(* Schneider Machine Expert - Basic project IC Flashing TM221CE40T, file version 2.7.0.0 *)
(* ProjectInformations: Name=New project *)

HARDWARE
  Cpu 0: TM221CE40T
  ModuleExtensionObject 0: TM3DI32K
  ModuleExtensionObject 1: TM3DQ32TK
  EthernetConfiguration: NetworkName=M221, IpAllocationMode=FixedAddress, IpAddress=192.168.0.2, SubnetMask=255.255.255.0
  SerialLineConfiguration: Baud=Baud19200, Parity=ParityEven, DataBits=DataBits8, StopBits=StopBits1, PhysicalMedium=PhysicalMediumRs485, TransmissionMode=TransmissionModeModbusRtu, SlaveId=1, Addressing=SlaveAddressing
  MastTask: UsePeriodScanMode=false, PeriodScan=100
  FastTask: Period=255
  CpuBehavior: StartingMode=StartAsPreviousState, AutoSaveRamOnEeprom=true, WatchdogPeriod=250

SYMBOLS  (address, symbol, comment, settings)
  %MW100:X14 TL_GREEN  "IO Output"
  %MW100:X15 TL_RED  "IO Output"
  %MW101:X1 BUZZER  "Output"
  %MW0:X4   ROBOT_PAUSE  "Input Robot1"
  %MW1:X6   IVACUM1  "Input Robot2"
  %M0         "M_START"
  %M1         "M_STOP"
  %M2         "M_CONTINUE"
  %M3         "M_PAUSE"
  %M4         "GRIPPER_ROTATE_CLOSE"
  %M5         "STATUS CB ON"
  %M6         "RELEASE_C_GRIPPER"
  %M7         "Reset"
  %M8         "Done"
  %M9         "Trig"
  %M10        "Start Read"
  %M11        "Start"
  %M12        "MANUAL"
  %M13        "Busy"
  %M14        "CB_RT"
  %M15        "DELAY_CUT_LEFT"
  %M16        "Cut Left"
  %M17        "Cut Right"
  %M19        "AUX_Seq_INIT"
  %M20        "Start_Write"
  %M21        "Abort"
  %M22        "Done_Write"
  %M23        "Busy_Write"
  %M24        "Aborted"
  %M25        "Error"
  %M26      MANUAL_GRIP_CLOSE  "M_Q4"
  %M27      SLIDER  "M_Q5"
  %M28        "M_Q6"
  %M29        "Manual Bowl"
  %M30        "EMG_Memory"
  %M31        "Start_Memory"
  %M47        "M_EMG"
  %M49        "POLARITY CHECKED"
  %M50        "NEGATIVE"
  %M51        "POSITIVE"
  %M52        "FIRST RUN"
  %M53        "DONE CUTTING"
  %M54        "NEGATIVE READY"
  %M55        "TRIGGER"
  %M56        "COUNTER OUTPUT"
  %M100       "Abort"
  %M102       "M_START"
  %S4       SB_TB10MS  "Time base of 10 ms generated by an internal clock"
  %S6       SB_TB1S  "Time base of 1 s generated by an internal clock"
  %MW0        "Input Robot1"
  %MW1        "Input Robot2"
  %MW100      "IO Output"
  %MW101      "Output"
  %TM2        "Left Cut"  [Preset=10, Base=TenMilliSeconds]
  %READ_VAR1   "READ OUTPUT ROBOT"  [Link(Value(FBComLinkParameterEnums=EthernetLink)), RemoteDeviceId(Value(int=1)), Timeout(Value(int=100)), ObjType(Value(FBComObjTypeParameterEnums=IW)), FirstObj(Value(int=31)), Quantity(Value(int=2)), IndexData(Value(int=100))]
  %WRITE_VAR0   [Link(Value(FBComLinkParameterEnums=EthernetLink)), RemoteDeviceId(Value(int=1)), Timeout(Value(int=100)), ObjType(Value(FBComObjTypeParameterEnums=MW)), FirstObj(Value(int=31)), Quantity(Value(int=2)), IndexData(Value(int=0))]
  %I0.0       "EMG"
  %I0.1       "PB START"
  %I0.2       "PB STOP"
  %I0.3       "PB Continue"
  %I0.4       "PB Pause"
  %I0.5       "Safety Relay"
  %I0.6       "Homing Sensor 1"
  %I0.7       "Homing Sensor 2"
  %I0.23      "iVacum1"
  %Q0.14      "TL Green"
  %Q0.15      "TL YelloW"
  %Q2.0       "TL Red"
  %Q2.1       "BUZZER"
  %Q2.2       "PB GREEN_LAMP"
  %Q2.3       "PB YELLOW_LAMP"
  %Q2.4       "PB RED_LAMP"

POU New POU
  (* SectionNumber=1 *)

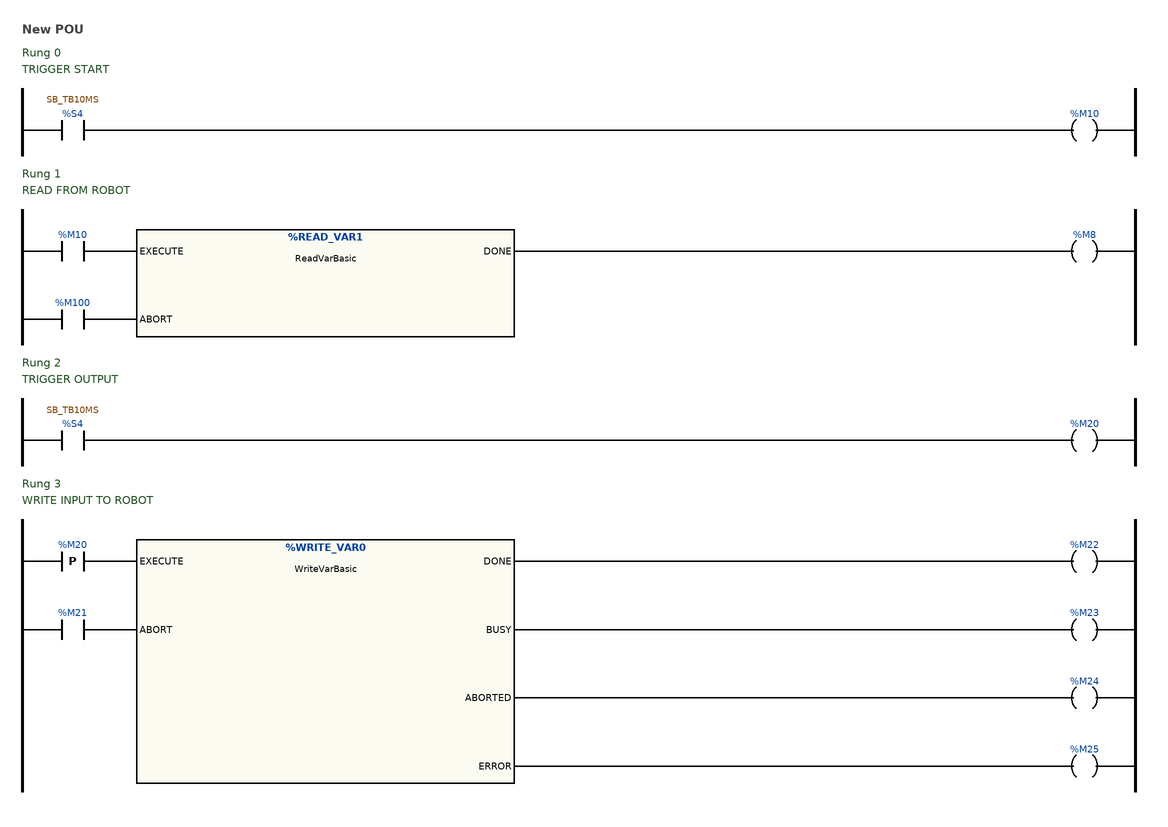

// Rung 0
// TRIGGER START
  LD %S4                  (* SB_TB10MS *)
  ST %M10
  // as ST:
  //   %M10 := SB_TB10MS;

// Rung 1
// READ FROM ROBOT
  BLK %READ_VAR1
  LD %M10
  EXECUTE
  LD %M100
  ABORT
  OUT_BLK
  LD DONE
  ST %M8
  END_BLK
  // as ST:
  //   %READ_VAR1(EXECUTE := %M10, ABORT := %M100);
  //   %M8 := %READ_VAR1.DONE;

// Rung 2
// TRIGGER OUTPUT
  LD %S4                  (* SB_TB10MS *)
  ST %M20
  // as ST:
  //   %M20 := SB_TB10MS;

// Rung 3
// WRITE INPUT TO ROBOT
  BLK %WRITE_VAR0
  LDR %M20
  EXECUTE
  LD %M21
  ABORT
  OUT_BLK
  LD DONE
  ST %M22
  LD BUSY
  ST %M23
  LD ABORTED
  ST %M24
  LD ERROR
  ST %M25
  END_BLK
  // as ST:
  //   %WRITE_VAR0(EXECUTE := RISING(%M20), ABORT := %M21);
  //   %M22 := %WRITE_VAR0.DONE;
  //   %M23 := %WRITE_VAR0.BUSY;
  //   %M24 := %WRITE_VAR0.ABORTED;
  //   %M25 := %WRITE_VAR0.ERROR;

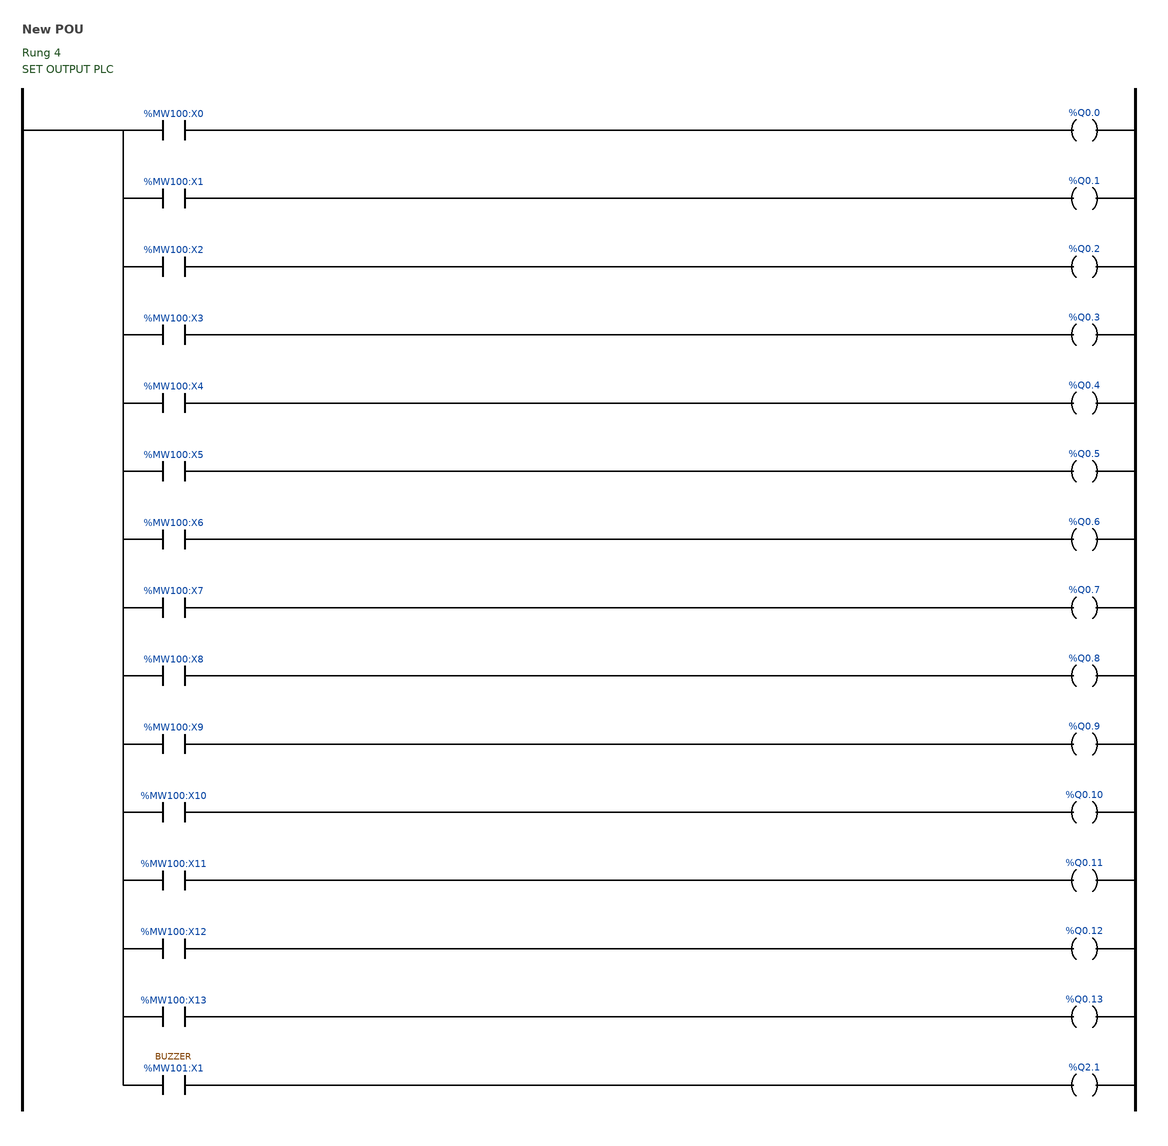

// Rung 4
// SET OUTPUT PLC
  LD 1
  MPS
  AND %MW100:X0
  ST %Q0.0
  MRD
  AND %MW100:X1
  ST %Q0.1
  MRD
  AND %MW100:X2
  ST %Q0.2
  MRD
  AND %MW100:X3
  ST %Q0.3
  MRD
  AND %MW100:X4
  ST %Q0.4
  MRD
  AND %MW100:X5
  ST %Q0.5
  MRD
  AND %MW100:X6
  ST %Q0.6
  MRD
  AND %MW100:X7
  ST %Q0.7
  MRD
  AND %MW100:X8
  ST %Q0.8
  MRD
  AND %MW100:X9
  ST %Q0.9
  MRD
  AND %MW100:X10
  ST %Q0.10
  MRD
  AND %MW100:X11
  ST %Q0.11
  MRD
  AND %MW100:X12
  ST %Q0.12
  MRD
  AND %MW100:X13
  ST %Q0.13
  MPP
  AND %MW101:X1
  ST %Q2.1
  // as ST:
  //   %Q0.0 := %MW100:X0;
  //   %Q0.1 := %MW100:X1;
  //   %Q0.2 := %MW100:X2;
  //   %Q0.3 := %MW100:X3;
  //   %Q0.4 := %MW100:X4;
  //   %Q0.5 := %MW100:X5;
  //   %Q0.6 := %MW100:X6;
  //   %Q0.7 := %MW100:X7;
  //   %Q0.8 := %MW100:X8;
  //   %Q0.9 := %MW100:X9;
  //   %Q0.10 := %MW100:X10;
  //   %Q0.11 := %MW100:X11;
  //   %Q0.12 := %MW100:X12;
  //   %Q0.13 := %MW100:X13;
  //   %Q2.1 := %MW101:X1;

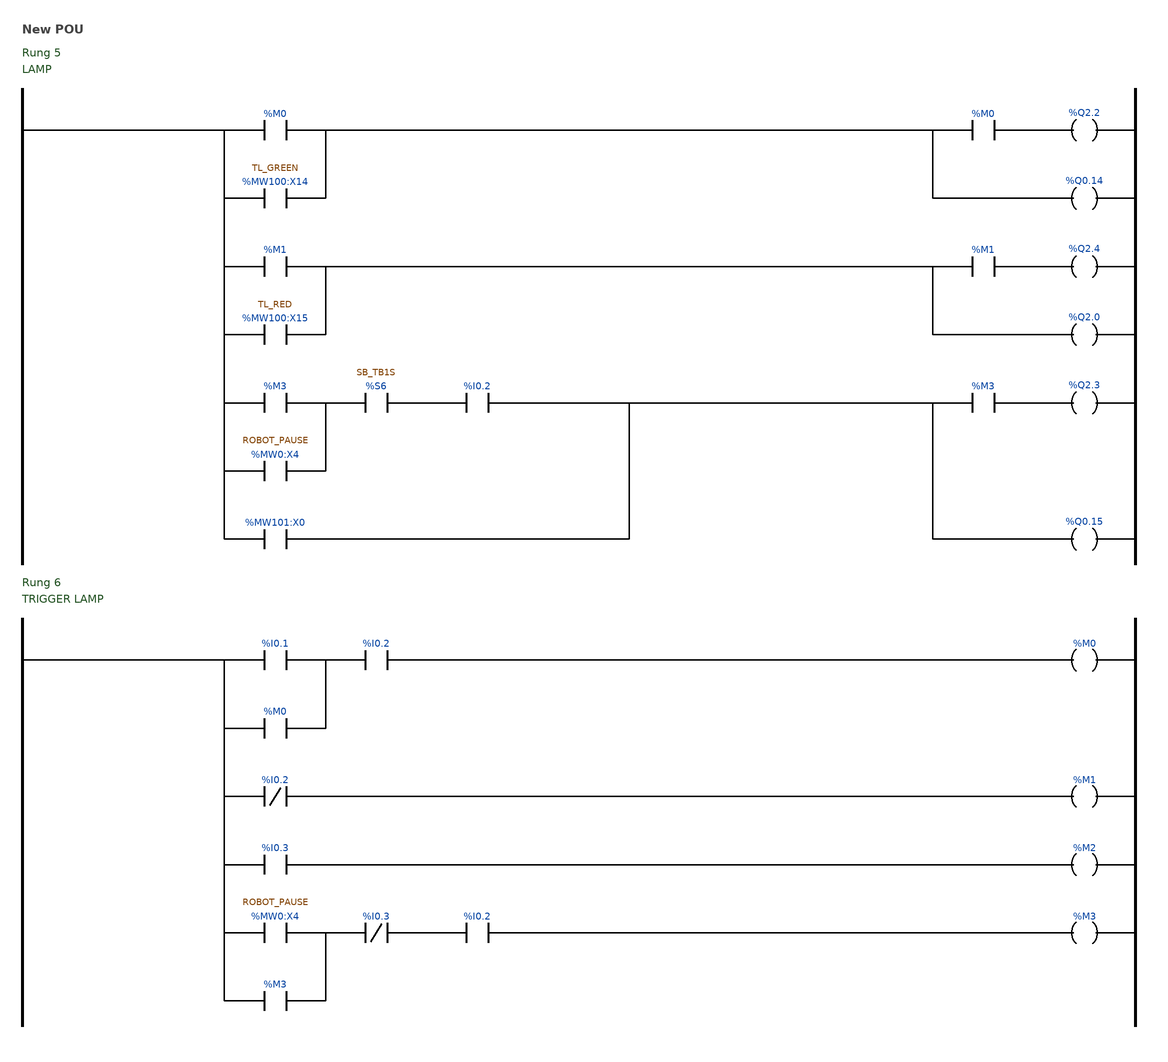

// Rung 5
// LAMP
  LD 1
  MPS
  AND( %M0
  OR %MW100:X14
  )
  MPS
  AND %M0
  ST %Q2.2
  MPP
  ST %Q0.14
  MRD
  AND( %M1
  OR %MW100:X15
  )
  MPS
  AND %M1
  ST %Q2.4
  MPP
  ST %Q2.0
  MPP
  AND( %M3
  OR %MW0:X4
  AND %S6                 (* SB_TB1S *)
  AND %I0.2
  OR %MW101:X0
  )
  MPS
  AND %M3
  ST %Q2.3
  MPP
  ST %Q0.15
  // as ST:
  //   %Q2.2 := (%M0 OR %MW100:X14) AND %M0;
  //   %Q0.14 := %M0 OR %MW100:X14;
  //   %Q2.4 := (%M1 OR %MW100:X15) AND %M1;
  //   %Q2.0 := %M1 OR %MW100:X15;
  //   %Q2.3 := ((%M3 OR %MW0:X4) AND SB_TB1S AND %I0.2 OR %MW101:X0) AND %M3;
  //   %Q0.15 := (%M3 OR %MW0:X4) AND SB_TB1S AND %I0.2 OR %MW101:X0;

// Rung 6
// TRIGGER LAMP
  LD 1
  MPS
  AND( %I0.1
  OR %M0
  )
  AND %I0.2
  ST %M0
  MRD
  ANDN %I0.2
  ST %M1
  MRD
  AND %I0.3
  ST %M2
  MPP
  AND( %MW0:X4
  OR %M3
  )
  ANDN %I0.3
  AND %I0.2
  ST %M3
  // as ST:
  //   %M0 := (%I0.1 OR %M0) AND %I0.2;
  //   %M1 := NOT %I0.2;
  //   %M2 := %I0.3;
  //   %M3 := (%MW0:X4 OR %M3) AND NOT %I0.3 AND %I0.2;

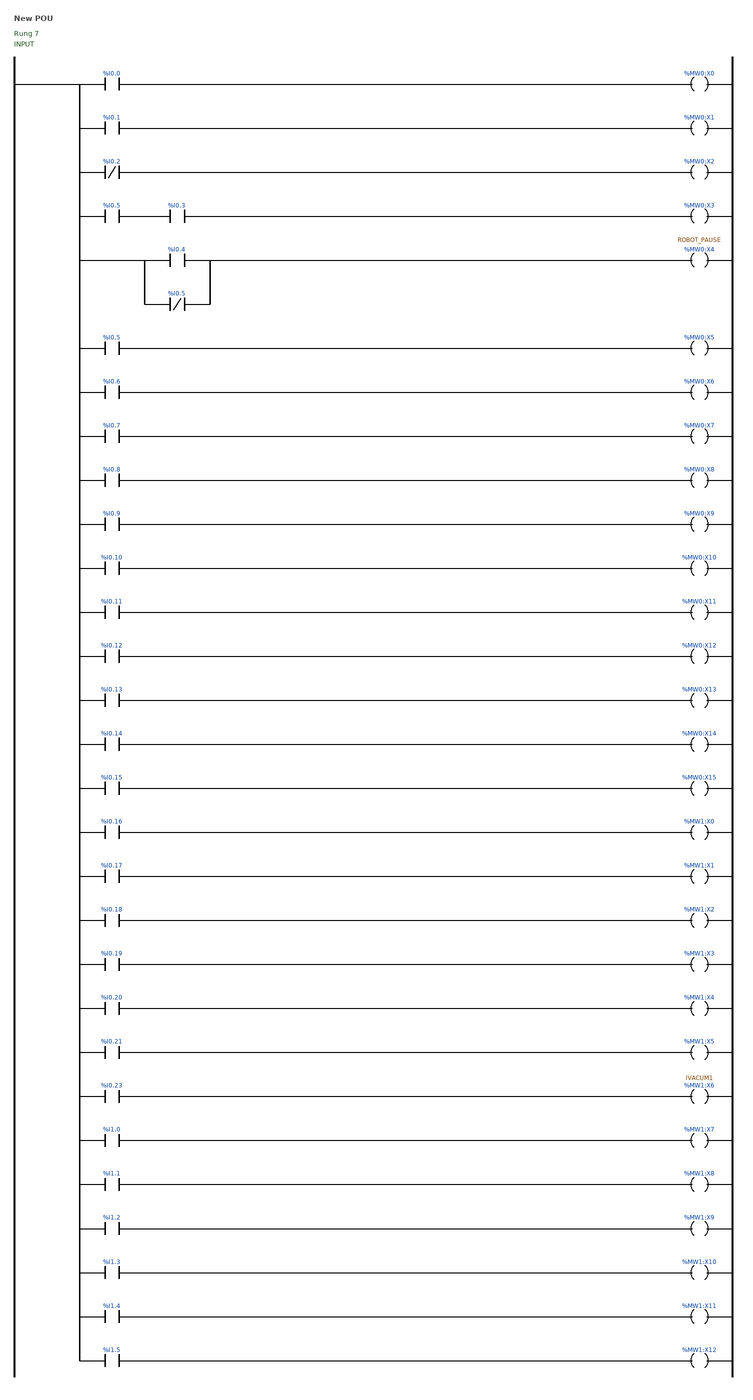

// Rung 7
// INPUT
  LD 1
  MPS
  AND %I0.0
  ST %MW0:X0
  MRD
  AND %I0.1
  ST %MW0:X1
  MRD
  ANDN %I0.2
  ST %MW0:X2
  MRD
  AND %I0.5
  AND %I0.3
  ST %MW0:X3
  MRD
  AND( %I0.4
  ORN %I0.5
  )
  ST %MW0:X4
  MRD
  AND %I0.5
  ST %MW0:X5
  MRD
  AND %I0.6
  ST %MW0:X6
  MRD
  AND %I0.7
  ST %MW0:X7
  MRD
  AND %I0.8
  ST %MW0:X8
  MRD
  AND %I0.9
  ST %MW0:X9
  MRD
  AND %I0.10
  ST %MW0:X10
  MRD
  AND %I0.11
  ST %MW0:X11
  MRD
  AND %I0.12
  ST %MW0:X12
  MRD
  AND %I0.13
  ST %MW0:X13
  MRD
  AND %I0.14
  ST %MW0:X14
  MRD
  AND %I0.15
  ST %MW0:X15
  MRD
  AND %I0.16
  ST %MW1:X0
  MRD
  AND %I0.17
  ST %MW1:X1
  MRD
  AND %I0.18
  ST %MW1:X2
  MRD
  AND %I0.19
  ST %MW1:X3
  MRD
  AND %I0.20
  ST %MW1:X4
  MRD
  AND %I0.21
  ST %MW1:X5
  MRD
  AND %I0.23
  ST %MW1:X6
  MRD
  AND %I1.0
  ST %MW1:X7
  MRD
  AND %I1.1
  ST %MW1:X8
  MRD
  AND %I1.2
  ST %MW1:X9
  MRD
  AND %I1.3
  ST %MW1:X10
  MRD
  AND %I1.4
  ST %MW1:X11
  MPP
  AND %I1.5
  ST %MW1:X12
  // as ST:
  //   %MW0:X0 := %I0.0;
  //   %MW0:X1 := %I0.1;
  //   %MW0:X2 := NOT %I0.2;
  //   %MW0:X3 := %I0.5 AND %I0.3;
  //   %MW0:X4 := %I0.4 OR NOT %I0.5;
  //   %MW0:X5 := %I0.5;
  //   %MW0:X6 := %I0.6;
  //   %MW0:X7 := %I0.7;
  //   %MW0:X8 := %I0.8;
  //   %MW0:X9 := %I0.9;
  //   %MW0:X10 := %I0.10;
  //   %MW0:X11 := %I0.11;
  //   %MW0:X12 := %I0.12;
  //   %MW0:X13 := %I0.13;
  //   %MW0:X14 := %I0.14;
  //   %MW0:X15 := %I0.15;
  //   %MW1:X0 := %I0.16;
  //   %MW1:X1 := %I0.17;
  //   %MW1:X2 := %I0.18;
  //   %MW1:X3 := %I0.19;
  //   %MW1:X4 := %I0.20;
  //   %MW1:X5 := %I0.21;
  //   %MW1:X6 := %I0.23;
  //   %MW1:X7 := %I1.0;
  //   %MW1:X8 := %I1.1;
  //   %MW1:X9 := %I1.2;
  //   %MW1:X10 := %I1.3;
  //   %MW1:X11 := %I1.4;
  //   %MW1:X12 := %I1.5;
